# EPICS substitutions: vacuumSimApp/Db/gauge.substitutions
# gauge substituion file

file db/gauge.db {
  pattern { G }
    { G1 }
    { G2 }
}
